Omron CX-Programmer project 新工程 (CX-Programmer 9.61)

# PLC 新PLC1: CP1E N30

## Global symbols (name address type ; comment)
0.00 BOOL  ; 启动开关
0.01 BOOL  ; M传感器
0.02 BOOL  ; H传感器
0.03 BOOL  ; L传感器
0.04 BOOL  ; 复位按钮
0.05 BOOL  ; 停止按钮
100.00 BOOL  ; A阀门
100.01 BOOL  ; B阀门
100.02 BOOL  ; 搅拌电机
100.03 BOOL  ; C阀门

## Program 新程序1 (cyclic task 0)

### Section 段1

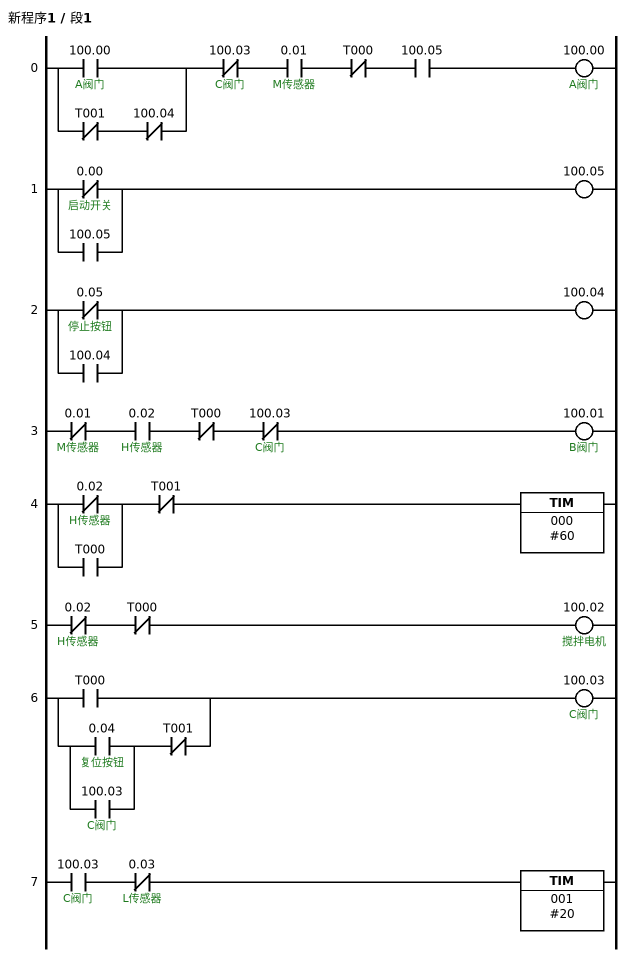
; rung 0
LD 100.00  ; A阀门
LDNOT T001
ANDNOT 100.04
ORLD
ANDNOT 100.03  ; C阀门
AND 0.01  ; M传感器
ANDNOT T000
AND 100.05
OUT 100.00  ; A阀门
; rung 1
LDNOT 0.00  ; 启动开关
OR 100.05
OUT 100.05
; rung 2
LDNOT 0.05  ; 停止按钮
OR 100.04
OUT 100.04
; rung 3
LDNOT 0.01  ; M传感器
AND 0.02  ; H传感器
ANDNOT T000
ANDNOT 100.03  ; C阀门
OUT 100.01  ; B阀门
; rung 4
LDNOT 0.02  ; H传感器
OR T000
ANDNOT T001
TIM 000 #60
; rung 5
LDNOT 0.02  ; H传感器
ANDNOT T000
OUT 100.02  ; 搅拌电机
; rung 6
LD T000
LD 0.04  ; 复位按钮
OR 100.03  ; C阀门
ANDNOT T001
ORLD
OUT 100.03  ; C阀门
; rung 7
LD 100.03  ; C阀门
ANDNOT 0.03  ; L传感器
TIM 001 #20
; rung 8
END(001)

### Section END
; rung 0
END(001)